INTERFACE I_Quantity EXTENDS I_Fallible


PROPERTY Units : T_MaxString
GET
END_GET
END_PROPERTY

END_INTERFACE

(* stored: Version 1.1.0.1
   Itf I_Quantity: Id {2968f420-eb06-4ec9-8610-471e30e82d60}
   Property Units: Id {68f968ed-7630-4d1a-a3e0-ed26644f9ec7}
   Get Get: Id {0e0a0f8f-9c5c-47f0-86a0-0f895a7ef1ea} *)
